// TIA Portal V19 export
TYPE "LUC_typeUnitModeStateTimes"
TITLE = LUC_typeUnitModeStateTimes
// Statistic of time spent in modes and states
// stored: Access Published
   STRUCT
      modeTimeCurrent { ExternalWritable := 'False'} : DInt;   // Actual time for current mode in seconds
      stateTimeCurrent { ExternalWritable := 'False'} : DInt;   // Actual time for current state in seconds
      accTimeSinceReset { ExternalWritable := 'False'} : DInt;   // Accumulated time since last reset in seconds
      actualTimeAllModes { ExternalWritable := 'False'} : Array[0.."LPMLV2022_MODES_UPPER_LIM"] of DInt;   // Actual time for all modes in seconds (former name: ModeCurrentTime)
      cumulativeTimeAllModes { ExternalWritable := 'False'} : Array[0.."LPMLV2022_MODES_UPPER_LIM"] of DInt;   // Cumulative time for all modes in seconds (former name: ModeCumulativeTime)
      actualTimeAllStatesOfAllModes { ExternalWritable := 'False'} : Array[0.."LPMLV2022_MODES_UPPER_LIM", 0.."LPMLV2022_STATES_UPPER_LIM"] of DInt;   // Actual time for all states in seconds (former name: StateCurrentTime)
      cumulativeTimeAllStatesOfAllModes { ExternalWritable := 'False'} : Array[0.."LPMLV2022_MODES_UPPER_LIM", 0.."LPMLV2022_STATES_UPPER_LIM"] of DInt;   // Cumulative time for all states in seconds (former name: StateCumulativeTime)
      actualTimeAllStatesOfCurrentMode { ExternalWritable := 'False'} : Array[0.."LPMLV2022_STATES_UPPER_LIM"] of DInt;   // Actual time for all states in current mode in seconds
      cumulativeTimeAllStatesOfCurrentMode { ExternalWritable := 'False'} : Array[0.."LPMLV2022_STATES_UPPER_LIM"] of DInt;   // Cumulative time for all states in current mode in seconds
      cumulativeTimeCurrentMode { ExternalWritable := 'False'} : DInt;   // Cumulative time for current mode in seconds
   END_STRUCT;
END_TYPE
